Staubli VAL3: SettingENC.dtx

num nCOLMAX = 39
num nCOLMIN
public num nColumn
public num nFocused
public num nListSize
num nROWMAX = 12
num nROWMIN
public num nRow
string sErrorMessage
string sErrorMsg[10]
  [1] = "An error has been detected in the Page library *\../*"
  [2] = "Variable sTxtBoxLen[*] has an illegal value"
  [3] = "Variable sTxtBoxPos[*] has an illegal value"
public string sFALSE = "FALSE"
public string sLabel[2]
  [0] = "-Encoder data ---"
  [1] = "- Filter ---"
public string sLabelPos[2]
  [0] = "0;0"
  [1] = "0;6"
public string sMenu = "; GENERAL ; ; DETECTION CONVEYOR ; Ok"
public string sTRUE = "TRUE"
public string sTitle
public string sTxtBoxAuthord[4]
  [0] = "0123456789"
  [1] = "0123456789"
  [2] = "0123456789."
  [3] = "0123456789."
public string sTxtBoxCaption[4]
  [0] = "LatchPeriod:"
  [1] = "Resolution :"
  [2] = "Length    : "
  [3] = "Delay(ms) : "
public string sTxtBoxLen[4]
  [0] = "2"
  [1] = "5"
  [2] = "3"
  [3] = "3"
public string sTxtBoxPos[4]
  [0] = "0;1"
  [1] = "0;2"
  [2] = "0;7"
  [3] = "0;8"
public string sTxtBoxRange[4]
  [0] = "0;99"
  [1] = "0;20000"
  [2] = "4;500"
  [3] = "1;20"
public string sTxtBoxType[4]
  [0] = "N"
  [1] = "N"
  [2] = "N"
  [3] = "D"
public string sTxtBoxVal[4]
  [0] = "1"
  [1] = "1024"
  [2] = "15"
  [3] = "0"
public string sListItem0
